TYPE HMIXTSMoverHelper_typ :
STRUCT
	BallImgVisibility:		BOOL;
	PlayerNumberVisibility: BOOL;
	PlayerNumber: 			UINT;
END_STRUCT
END_TYPE

(* stored: Version 1.1.0.1, ProductVersion 3.1.4024.12
   DUT HMIXTSMoverHelper_typ: Id {3e490a70-6328-0a90-3608-650dbf2daa58} *)
